# EPICS substitutions: db/EL3024.substitutions
file EL3024.template
{ 	pattern
	{
		TERMINAL,
		DESC1,	SCAN1,	ADEL1,	EGUF1,	EGUL1,	HIGH1,	HIHI1,	HOPR1,	HYST1,	LOLO1,	LOPR1,	LOW1,	MDEL1,	SMOO1,	UNIT1,
		DESC2,	SCAN2,	ADEL2,	EGUF2,	EGUL2,	HIGH2,	HIHI2,	HOPR2,	HYST2,	LOLO2,	LOPR2,	LOW2,	MDEL2,	SMOO2,	UNIT2,
		DESC3,	SCAN3,	ADEL3,	EGUF3,	EGUL3,	HIGH3,	HIHI3,	HOPR3,	HYST3,	LOLO3,	LOPR3,	LOW3,	MDEL3,	SMOO3,	UNIT3,
		DESC4,	SCAN4,	ADEL4,	EGUF4,	EGUL4,	HIGH4,	HIHI4,	HOPR4,	HYST4,	LOLO4,	LOPR4,	LOW4,	MDEL4,	SMOO4,	UNIT4
	}
	{
	}
}
